TYPE ST_PumpErrors :
STRUCT	
	Thermal			: BOOL;
END_STRUCT
END_TYPE

(* stored: Version 1.1.0.1, ProductVersion 3.1.4020.12
   DUT ST_PumpErrors: Id {b900ef99-01d9-4060-a648-784aa27acd56} *)
